Universal Robots PolyScope program: cottonMachineOn.urp

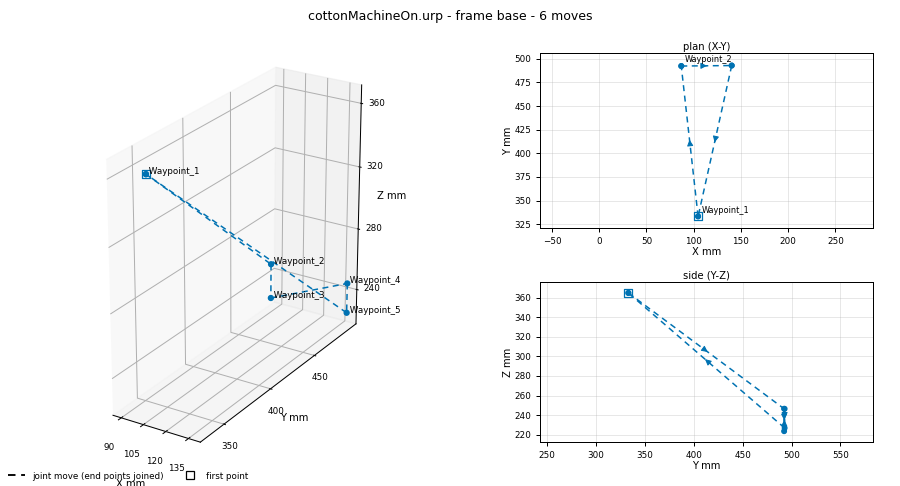
[picture p0: tool path of cottonMachineOn.urp in frame base, 6 of 8 moves have a stored position in this frame; points joined in program order, loops and branches not executed]
Program cottonMachineOn (installation=default directory=/programs/DavidMelin createdIn=5.12.4.1101661 lastSavedIn=5.12.4.1101661 robotSerialNumber=20225502378)
Calibrated DH parameters: a=[0.00022, -0.425328, -0.389701, 0.000059, 0.000065, 0]; d=[0.162608, 0.803456, 9.992211, -10.662202, 0.099702, 0.099559]; alpha=[1.570756, 0.001543, 0.004316, 1.570651, -1.570122, 0]; deltaTheta=[0, 0.002917, 0.116094, -0.119008, 0, -0.000001]
Robot Program (runOnlyOnce=true)
  MoveJ speed 60 deg/s, acceleration 80 deg/s^2 (useActiveTCP=true) feature=Base
    Waypoint Waypoint (Variable): variable=cotonHomePos
  URCap Gripper (Robotiq_Grippers, Robotiq Inc.) dataModel(position=100.0, force=0.0, speed=100.0, positionInDouble=100.0, forceInDouble=0.0, speedInDouble=100.0, slaveIds=[9], blocking=true)
  MoveJ speed 60 deg/s, acceleration 80 deg/s^2 (useActiveTCP=true) feature=Base
    Waypoint Waypoint_1: TCP in base x=104.659 y=333.276 z=364.782 mm, rx=-2.4906 ry=0.0958 rz=-0.1132 rad; joints [98.535, -64.728, -139.703, -29.68, 79.086, 9.45] deg
    Waypoint Waypoint_2: TCP in base x=86.854 y=492.403 z=246.454 mm, rx=-2.395 ry=0.1183 rz=-0.0956 rad; joints [97.806, -104.935, -129.813, 6.212, 78.977, 9.441] deg
    Waypoint Waypoint_3: TCP in base x=86.863 y=492.414 z=223.527 mm, rx=-2.3949 ry=0.1183 rz=-0.0956 rad; joints [97.803, -108.318, -130.629, 10.412, 78.962, 9.444] deg
    Waypoint Waypoint_4: TCP in base x=140.276 y=492.921 z=246.4 mm, rx=-2.3951 ry=0.1183 rz=-0.0956 rad; joints [90.496, -106.571, -127.634, 6.506, 83.868, 3.943] deg
    Waypoint Waypoint_5: TCP in base x=140.246 y=492.94 z=226.795 mm, rx=-2.395 ry=0.1182 rz=-0.0956 rad; joints [90.498, -109.344, -128.315, 9.965, 83.856, 3.945] deg
    Waypoint Waypoint_6: TCP in base x=104.69 y=333.274 z=364.784 mm, rx=-2.4906 ry=0.0959 rz=-0.1132 rad; joints [98.529, -64.729, -139.702, -29.68, 79.085, 9.45] deg
    Waypoint Waypoint (Variable): variable=cotonHomePos
